(* IEC 61131-3 sources: programs/VI-54/VI-54_20171205/VI-54_20171205/Stations/Screen/LseClass170718/Class/DiagnosticUserFunction, 1 file *)

(* ---- DiagnosticUserFunction.st ---- *)
(*!
<Class
	Name               = "DiagnosticUserFunction"
	Revision           = "1.0"
	RealtimeTask       = "false"
	CyclicTask         = "false"
	BackgroundTask     = "false"
	Sigmatek           = "false"
	OSInterface        = "false"
	HighPriority       = "false"
	Automatic          = "false"
	UpdateMode         = "Prescan"
	SharedCommandTable = "true"
	Objectsize         = "(284,120)"
	Comment            = "Use this class as base class for new functions.">
	<Channels>
		<Server Name="sStatus" Visualized="false" Initialize="false" WriteProtected="true" Retentive="false" Comment="Actual status."/>
		<Client Name="cSigCLib" Required="false" Internal="false" Comment="Object channel to SigCLib. Does not have to be connected."/>
	</Channels>
	<RevDoku>
		<Owner Company="Sigmatek"/>
		<Dokumentation Revision="1.0" Date="2016-06-02" Author="HötAnt" Company="Sigmatek" Description="Creation"/>
	</RevDoku>
</Class>
*)
DiagnosticUserFunction : CLASS
  //Servers:
	sStatus 	: SvrChCmd_iprStates;
  //Clients:
	cSigCLib 	: CltChCmd_SigCLib;
  //Variables:
		Fault 	: _DiagErrorCode;
  //Functions:
				//! <Function Comment="Use this method to set the drive path." Name="SetDrivePath"/>
	FUNCTION VIRTUAL GLOBAL SetDrivePath
		VAR_INPUT
			pDP 	: ^CHAR;			//! <Variable Comment="Pointer to the data with the drive path." Name="SetDrivePath.pDP"/>
		END_VAR;
				//! <Function Comment="Receive data." Name="ReceivedData"/>
	FUNCTION VIRTUAL GLOBAL ReceivedData
		VAR_INPUT
			size 	: UDINT;			//! <Variable Comment="Size of the received data." Name="ReceivedData.size"/>
			pdata 	: ^USINT;			//! <Variable Comment="Pointer to the received data." Name="ReceivedData.pdata"/>
			OptCMD 	: USINT;			//! <Variable Comment="Optional command." Name="ReceivedData.OptCMD"/>
		END_VAR
		VAR_OUTPUT
			retcode 	: BOOL;			//! <Variable Comment="FALSE..Error&#13;&#10;TRUE..Data received" Name="ReceivedData.retcode"/>
		END_VAR;
				//! <Function Comment="This method will be called cyclic when the diagnostic export is started." Name="WorkMethode"/>
	FUNCTION VIRTUAL GLOBAL WorkMethode;
				//! <Function Comment="Get the actual state." Name="GetWorkState"/>
	FUNCTION VIRTUAL GLOBAL GetWorkState
		VAR_OUTPUT
			retcode 	: iprStates;			//! <Variable Comment="Actual state." Name="GetWorkState.retcode"/>
		END_VAR;
				//! <Function Comment="Get error code." Name="GetErrorCode"/>
	FUNCTION VIRTUAL GLOBAL GetErrorCode
		VAR_OUTPUT
			retcode 	: _DiagErrorCode;			//! <Variable Comment="Error code." Name="GetErrorCode.retcode"/>
		END_VAR;
				//! <Function Comment="Is called when the work method finished." Name="EndWork"/>
	FUNCTION VIRTUAL GLOBAL EndWork;
  //Tables:
	FUNCTION @STD
		VAR_OUTPUT
			ret_code	: CONFSTATES;
		END_VAR;
	FUNCTION GLOBAL TAB @CT_;
END_CLASS;

#pragma usingLtd SigCLib

#pragma warning(disable:73);
#pragma warning(disable:76);
FUNCTION VIRTUAL GLOBAL DiagnosticUserFunction::WorkMethode

END_FUNCTION

FUNCTION VIRTUAL GLOBAL DiagnosticUserFunction::GetWorkState
	VAR_OUTPUT
		retcode 	: iprStates;
	END_VAR

END_FUNCTION

FUNCTION VIRTUAL GLOBAL DiagnosticUserFunction::GetErrorCode
	VAR_OUTPUT
		retcode 	: _DiagErrorCode;
	END_VAR

  retcode := Fault;

END_FUNCTION

FUNCTION VIRTUAL GLOBAL DiagnosticUserFunction::ReceivedData
	VAR_INPUT
		size 	: UDINT;
		pdata 	: ^USINT;
		OptCMD 	: USINT;
	END_VAR
	VAR_OUTPUT
		retcode 	: BOOL;
	END_VAR

END_FUNCTION

FUNCTION VIRTUAL GLOBAL DiagnosticUserFunction::EndWork

END_FUNCTION

FUNCTION VIRTUAL GLOBAL DiagnosticUserFunction::SetDrivePath
	VAR_INPUT
		pDP 	: ^CHAR;
	END_VAR

END_FUNCTION

#pragma warning(default:73);
#pragma warning(default:76);
